# B&R Automation Studio project PO_MiRTS_Lab1
Automation Studio 4.5.2.102

## Configuration Config1

### Task classes (Cpu.sw)
```
Cyclic#4:
  Program <- Program.prg
Binaries: udbdef, TCData, ashwac, arconfig, asfw, ashwd, iomap, User, Role, sysconf
Libraries: MotorCtrl
```

### Hardware
```
4PP065_0351_P74 : 4PP065.0351-P74 v1.0.4.0
  Connector IF5:
    ActivateDevice = 1
  ConfigurationID = lab1_Config1
  Simulation = 1
  KeyMappingFile = VC\4PP065_0351_P74.dis
```

## Logical view

Binary libraries used (declarations not repeated): operator, runtime, astime, AsIecCon

### Library Logical/Libraries/MotorCtrl (ANSIC)

#### MotorCtrl.fun - Exported functions and function blocks
```iecst
{REDUND_ERROR} {REDUND_UNREPLICABLE} FUNCTION_BLOCK FB_Motor (*TODO: Add your comment here*) (*$GROUP=User,$CAT=User,$GROUPICON=User.png,$CATICON=User.png*)
	VAR_INPUT
		u : {REDUND_UNREPLICABLE} REAL;
	END_VAR
	VAR_OUTPUT
		out_w : {REDUND_UNREPLICABLE} REAL;
	END_VAR
	VAR
		integrator : {REDUND_UNREPLICABLE} FB_Integrator;
		Tm : {REDUND_UNREPLICABLE} REAL;
		ke : {REDUND_UNREPLICABLE} REAL;
		dt : {REDUND_UNREPLICABLE} REAL;
	END_VAR
END_FUNCTION_BLOCK

{REDUND_ERROR} {REDUND_UNREPLICABLE} FUNCTION_BLOCK FB_Integrator (*TODO: Add your comment here*) (*$GROUP=User,$CAT=User,$GROUPICON=User.png,$CATICON=User.png*)
	VAR_INPUT
		in : {REDUND_UNREPLICABLE} REAL;
	END_VAR
	VAR_OUTPUT
		out : {REDUND_UNREPLICABLE} REAL;
	END_VAR
	VAR
		dt : {REDUND_UNREPLICABLE} REAL;
		state : {REDUND_UNREPLICABLE} REAL;
	END_VAR
END_FUNCTION_BLOCK

{REDUND_ERROR} {REDUND_UNREPLICABLE} FUNCTION_BLOCK FB_Regulator (*TODO: Add your comment here*) (*$GROUP=User,$CAT=User,$GROUPICON=User.png,$CATICON=User.png*)
	VAR_INPUT
		e : {REDUND_UNREPLICABLE} REAL;
	END_VAR
	VAR_OUTPUT
		u : {REDUND_UNREPLICABLE} REAL;
	END_VAR
	VAR
		k_p : {REDUND_UNREPLICABLE} REAL;
		k_i : {REDUND_UNREPLICABLE} REAL;
		integrator : {REDUND_UNREPLICABLE} FB_Integrator;
		iyOld : {REDUND_UNREPLICABLE} REAL;
		max_abs_value : {REDUND_UNREPLICABLE} REAL;
		dt : {REDUND_UNREPLICABLE} REAL;
	END_VAR
END_FUNCTION_BLOCK
```

#### FB_Motor.c
```c
#include <bur/plctypes.h>
#ifdef __cplusplus
	extern "C"
	{
#endif
	#include "MotorCtrl.h"
#ifdef __cplusplus
	};
#endif
/* TODO: Add your comment here */
void FB_Motor(struct FB_Motor* inst)
{
	/*TODO: Add your code here*/
	REAL a = inst->u / inst->ke - inst->out_w;
	REAL b = a / inst->Tm;

	inst->integrator.in = b;
	FB_Integrator(&inst->integrator);

	inst->out_w = inst->integrator.out;
}
```

#### FB_Regulator.c
```c
#include <bur/plctypes.h>
#ifdef __cplusplus
	extern "C"
	{
#endif
	#include "MotorCtrl.h"
#ifdef __cplusplus
	};
#endif
/* TODO: Add your comment here */
void FB_Regulator(struct FB_Regulator* inst)
{
	/*TODO: Add your code here*/
	REAL a = inst->e * inst->k_p;
	REAL b = inst->e * inst->k_i; //inst->dt
	a = a > inst->max_abs_value ? inst->max_abs_value : a;
	a = a < -inst->max_abs_value ? -inst->max_abs_value : a;
	inst->integrator.in = b + inst->iyOld;
	FB_Integrator(&inst->integrator);
	REAL sum = a + inst->integrator.out;
	inst->u = sum;
	inst->u = inst->u > inst->max_abs_value ? inst->max_abs_value : inst->u;
	inst->u = inst->u < -inst->max_abs_value ? -inst->max_abs_value : inst->u;
	inst->iyOld = inst->u - sum;
}
```

### Program Logical/Program

#### Variables.var
```iecst
VAR
	counter1 : REAL;
	fb_regulator : FB_Regulator;
	speed : REAL;
	fb_motor : FB_Motor;
	enable : BOOL := TRUE;
	fb_motor2 : FB_Motor;
	counter : REAL;
END_VAR
```

#### Cyclic.c
```c
#include <bur/plctypes.h>

#ifdef _DEFAULT_INCLUDES
	#include <AsDefault.h>
#endif

void _CYCLIC ProgramCyclic(void)
{
	if (enable)
	{
		if (counter == 200)
		{
			speed = 0;
			counter++;
		}
		else if (counter == 50)
		{
			speed = 50;
		}
		if (counter < 201)
			counter++;

		fb_regulator.e = speed + fb_motor.out_w;
		FB_Regulator(&fb_regulator);
		fb_motor.u = fb_regulator.u;
		fb_motor2.u = speed * fb_motor2.ke;
		FB_Motor(&fb_motor);
		FB_Motor(&fb_motor2);
	}
}
```

#### Init.c
```c
#include <bur/plctypes.h>

#ifdef _DEFAULT_INCLUDES
	#include <AsDefault.h>
#endif

void _INIT ProgramInit(void)
{
	fb_motor.dt = 0.01;
	fb_motor.ke = 0.24;
	fb_motor.Tm = 0.1;
	fb_motor.u = 0;
	fb_motor.integrator.dt = 0.01;

	fb_motor2.dt = 0.01;
	fb_motor2.ke = 0.24;
	fb_motor2.Tm = 0.1;
	fb_motor2.u = 0;
	fb_motor2.integrator.dt = 0.01;

	fb_regulator.dt = 0.01;
	fb_regulator.integrator.dt = 0.01;
	fb_regulator.k_i = 7.2;
	fb_regulator.k_p = 0.24 * 3;
	fb_regulator.max_abs_value = 24.0;

	speed = 0;
	counter = 0;

}
```

Listed in the project but not available here: Logical/Libraries/MotorCtrl/Types.typ, Logical/Libraries/MotorCtrl/Constants.var, Logical/Libraries/MotorCtrl/FB_Integrator.c
